FUNCTION_BLOCK FB_Selettore_Colori
VAR_INPUT
END_VAR
VAR_OUTPUT
END_VAR
VAR
END_VAR

END_FUNCTION_BLOCK

(* stored: Version 1.1.0.1, ProductVersion 3.1.4024.12
   POU FB_Selettore_Colori: Id {5352a273-edff-4dd4-83d4-c79be356614d}, SpecialFunc None *)
